// Mitsubishi GX Works2 project: PLC_group4 (1)   PLC: FX3G

// global labels: Global1
VAR_GLOBAL
  Start_Day_Switch AT X007 : BOOL;
  Oat_input AT D1110 : REAL;
  Oat_On_Hand AT D1120 : REAL;
  Protein_input AT D1130 : REAL;
  Protein_On_Hand AT D1140 : REAL;
  Honey_input AT D1150 : REAL;
  Honey_On_Hand AT D1160 : REAL;
END_VAR
VAR_GLOBAL CONSTANT
  Oat_LB : REAL := 400.0;
  Honey_LB : REAL := 160.0;
END_VAR
VAR_GLOBAL
  Ready_for_production AT M0 : BOOL;
  Emergency_Switch AT X005 : BOOL;
  Day_On AT Y000 : BOOL;
  Choose_Type AT X003 : BOOL;
  Analog_input1 AT D8280 : INT;
END_VAR
VAR_GLOBAL CONSTANT
  divide_input : REAL := 400.0;
  Protein_LB1 : REAL := 320.0;
END_VAR
VAR_GLOBAL
  Analog1_value AT D1170 : REAL;
END_VAR
VAR_GLOBAL CONSTANT
  Protein_type_LB : REAL := 5;
END_VAR
VAR_GLOBAL
  Protein_indicator AT M4 : BOOL;
END_VAR
VAR_GLOBAL CONSTANT
  Calssic_type_UB : REAL := 5.0;
END_VAR
VAR_GLOBAL
  Classic_indicator AT M5 : BOOL;
END_VAR
VAR_GLOBAL CONSTANT
  Oat_Classic_LB : REAL := 400.0;
  Protein_pro_LB1 : REAL := 320.0;
  Honey_pro_LB : REAL := 160.0;
END_VAR
VAR_GLOBAL
  Flag_oatClassic_production AT M1 : BOOL;
  Flag_proteinPro_production AT M2 : BOOL;
  Flag_honeyPro_production AT M3 : BOOL;
END_VAR
VAR_GLOBAL CONSTANT
  Protein_Calssic_LB : REAL := 160.0;
END_VAR
VAR_GLOBAL
  Flag_proteinClassic_production AT M6 : BOOL;
END_VAR
VAR_GLOBAL CONSTANT
  Honey_Classic_LB : REAL := 120.0;
END_VAR
VAR_GLOBAL
  Flag_HoneyClassic_production AT M7 : BOOL;
  Classic_check AT M8 : BOOL;
END_VAR
VAR_GLOBAL CONSTANT
  Oat_protein_LB : REAL := 240.0;
END_VAR
VAR_GLOBAL
  Flag_oatPro_production AT M9 : BOOL;
  Pro_check AT M10 : BOOL;
  TimerPro AT TC1 : BOOL;
  TV_5sec AT K50 : WORD;
  Mixing AT Y003 : BOOL;
  Stat_mix AT TS1 : BOOL;
  Analog_Output1 AT D8282 : INT;
  energy_bar_amount AT D1100 : REAL;
END_VAR
VAR_GLOBAL CONSTANT
  Mix_Classic : REAL := 680;
END_VAR
VAR_GLOBAL
  Mix_Total AT D1190 : REAL;
END_VAR
VAR_GLOBAL CONSTANT
  Mix_Pro : REAL := 720;
END_VAR
VAR_GLOBAL
  Start_Cooking AT X002 : BOOL;
  finish_cooking AT M11 : BOOL;
  help_cook AT M12 : BOOL;
  TC_2 AT TC2 : BOOL;
  blinkTime AT K5 : WORD;
  TS_2 AT TS2 : BOOL;
  Y_1 AT Y001 : BOOL;
  TC_3 AT TC3 : BOOL;
  TS_3 AT TS3 : BOOL;
  Y_2 AT Y002 : BOOL;
  TC_4 AT TC4 : BOOL;
  Classic_Time AT K40 : WORD;
  Protein_Time AT K50 : WORD;
  TC_5 AT TC5 : BOOL;
  Cooking_Tot AT D1200 : REAL;
  TS_4 AT TS4 : BOOL;
  TS_5 AT TS5 : BOOL;
  Start_pack AT X006 : BOOL;
  This_pack AT X000 : BOOL;
  One_packed AT K1 : WORD;
  One_start AT CC1 : BOOL;
  Eight_end AT CC2 : BOOL;
  Eight_packed AT K8 : WORD;
  Add_pack AT CS1 : BOOL;
  Last_pack AT CS2 : BOOL;
  Pack_inProcess AT Y004 : BOOL;
  Total_packges AT D1210 : REAL;
  Add_packge AT E1.0 : REAL;
END_VAR
VAR_GLOBAL CONSTANT
  Change_to_double : REAL := 40.0;
END_VAR
VAR_GLOBAL
  TS_1 AT TS1 : BOOL;
  finish_mix AT M13 : BOOL;
END_VAR

// task Task_01 (event TRUE, interval 0, priority 31): POU_01

PROGRAM POU_01
VAR CONSTANT
  Protein_LB : REAL := 320.0;
END_VAR
VAR
  analog_output : WORD;
END_VAR
(* structured ladder/FBD written out as ST: instructions are called as NAME(EN, inputs, outputs); _pN, _eN, _tN stand for wires *)
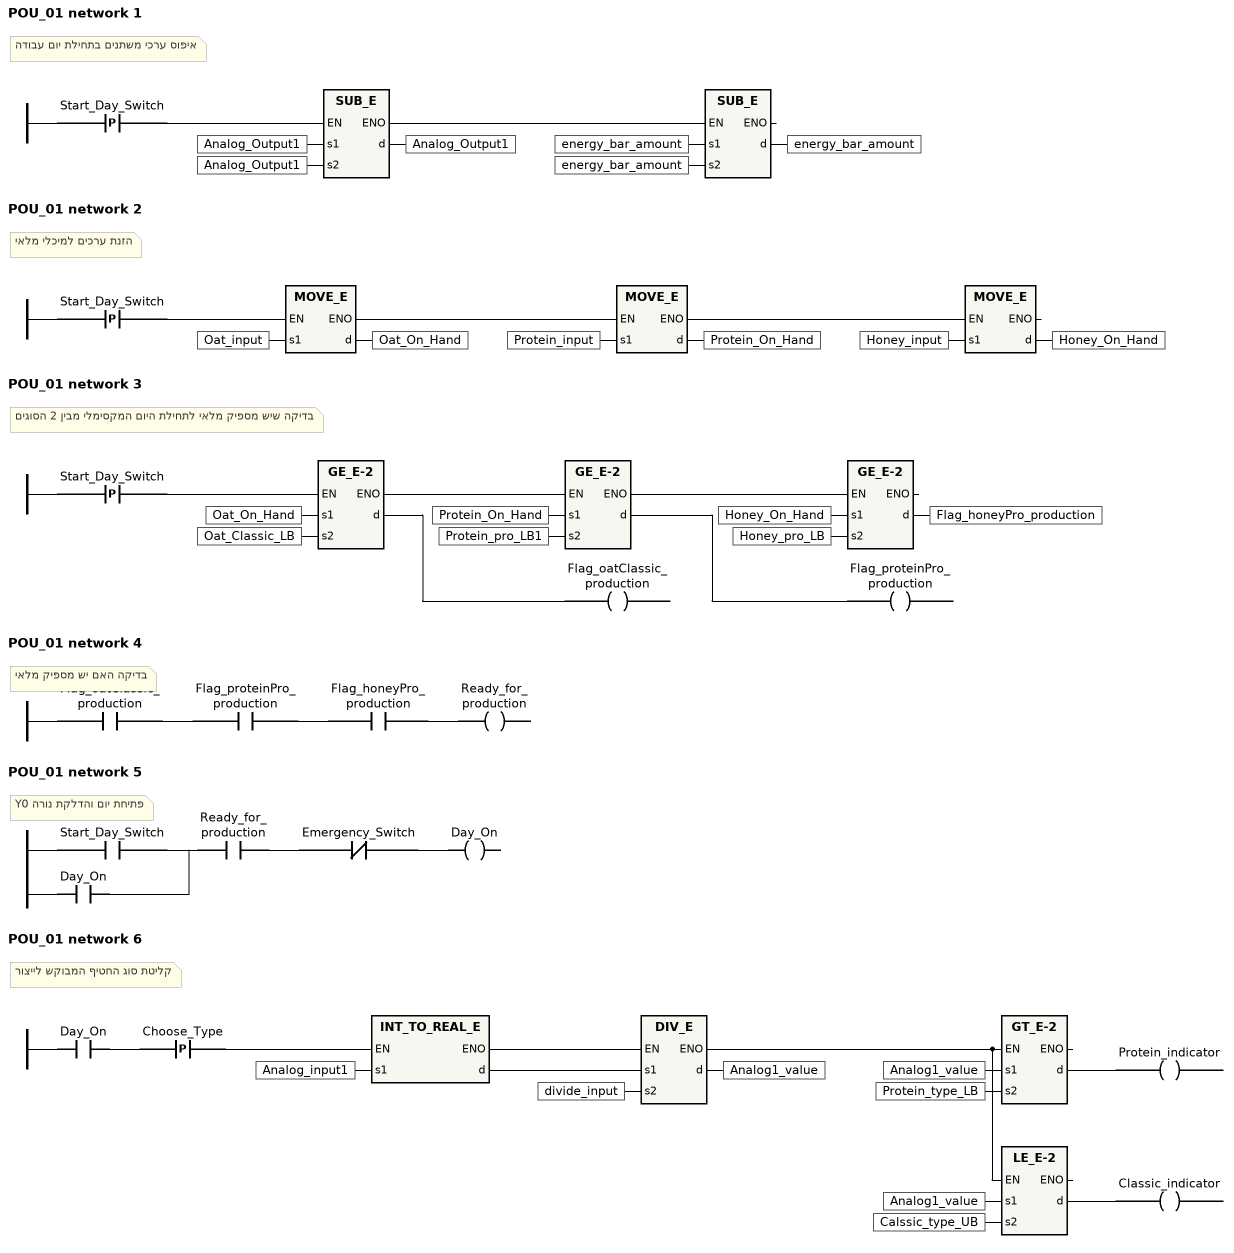
(* network 1 *)
(* איפוס ערכי משתנים בתחילת יום עבודה *)
_e1 := SUB_E(LDP(TRUE, Start_Day_Switch), Analog_Output1, Analog_Output1, Analog_Output1);
SUB_E(_e1, energy_bar_amount, energy_bar_amount, energy_bar_amount);
(* network 2 *)
(* הזנת ערכים למיכלי מלאי *)
_e1 := MOVE_E(LDP(TRUE, Start_Day_Switch), Oat_input, Oat_On_Hand);
_e2 := MOVE_E(_e1, Protein_input, Protein_On_Hand);
MOVE_E(_e2, Honey_input, Honey_On_Hand);
(* network 3 *)
(* בדיקה שיש מספיק מלאי לתחילת היום המקסימלי מבין 2 הסוגים *)
_e2 := GE_E(LDP(TRUE, Start_Day_Switch), Oat_On_Hand, Oat_Classic_LB, _t1);
_e4 := GE_E(_e2, Protein_On_Hand, Protein_pro_LB1, _t3);
GE_E(_e4, Honey_On_Hand, Honey_pro_LB, Flag_honeyPro_production);
Flag_oatClassic_production := _t1;
Flag_proteinPro_production := _t3;
(* network 4 *)
(* בדיקה האם יש מספיק מלאי *)
Ready_for_production := Flag_oatClassic_production AND Flag_proteinPro_production AND Flag_honeyPro_production;
(* network 5 *)
(* פתיחת יום והדלקת נורה Y0 *)
Day_On := ((Start_Day_Switch OR Day_On) AND Ready_for_production) AND NOT Emergency_Switch;
(* network 6 *)
(* קליטת סוג החטיף המבוקש לייצור *)
_e2 := INT_TO_REAL_E(Day_On AND LDP(TRUE, Choose_Type), Analog_input1, _t1);
_e3 := DIV_E(_e2, _t1, divide_input, Analog1_value);
GT_E(_e3, Analog1_value, Protein_type_LB, _t4);
Protein_indicator := _t4;
LE_E(_e3, Analog1_value, Calssic_type_UB, _t5);
Classic_indicator := _t5;
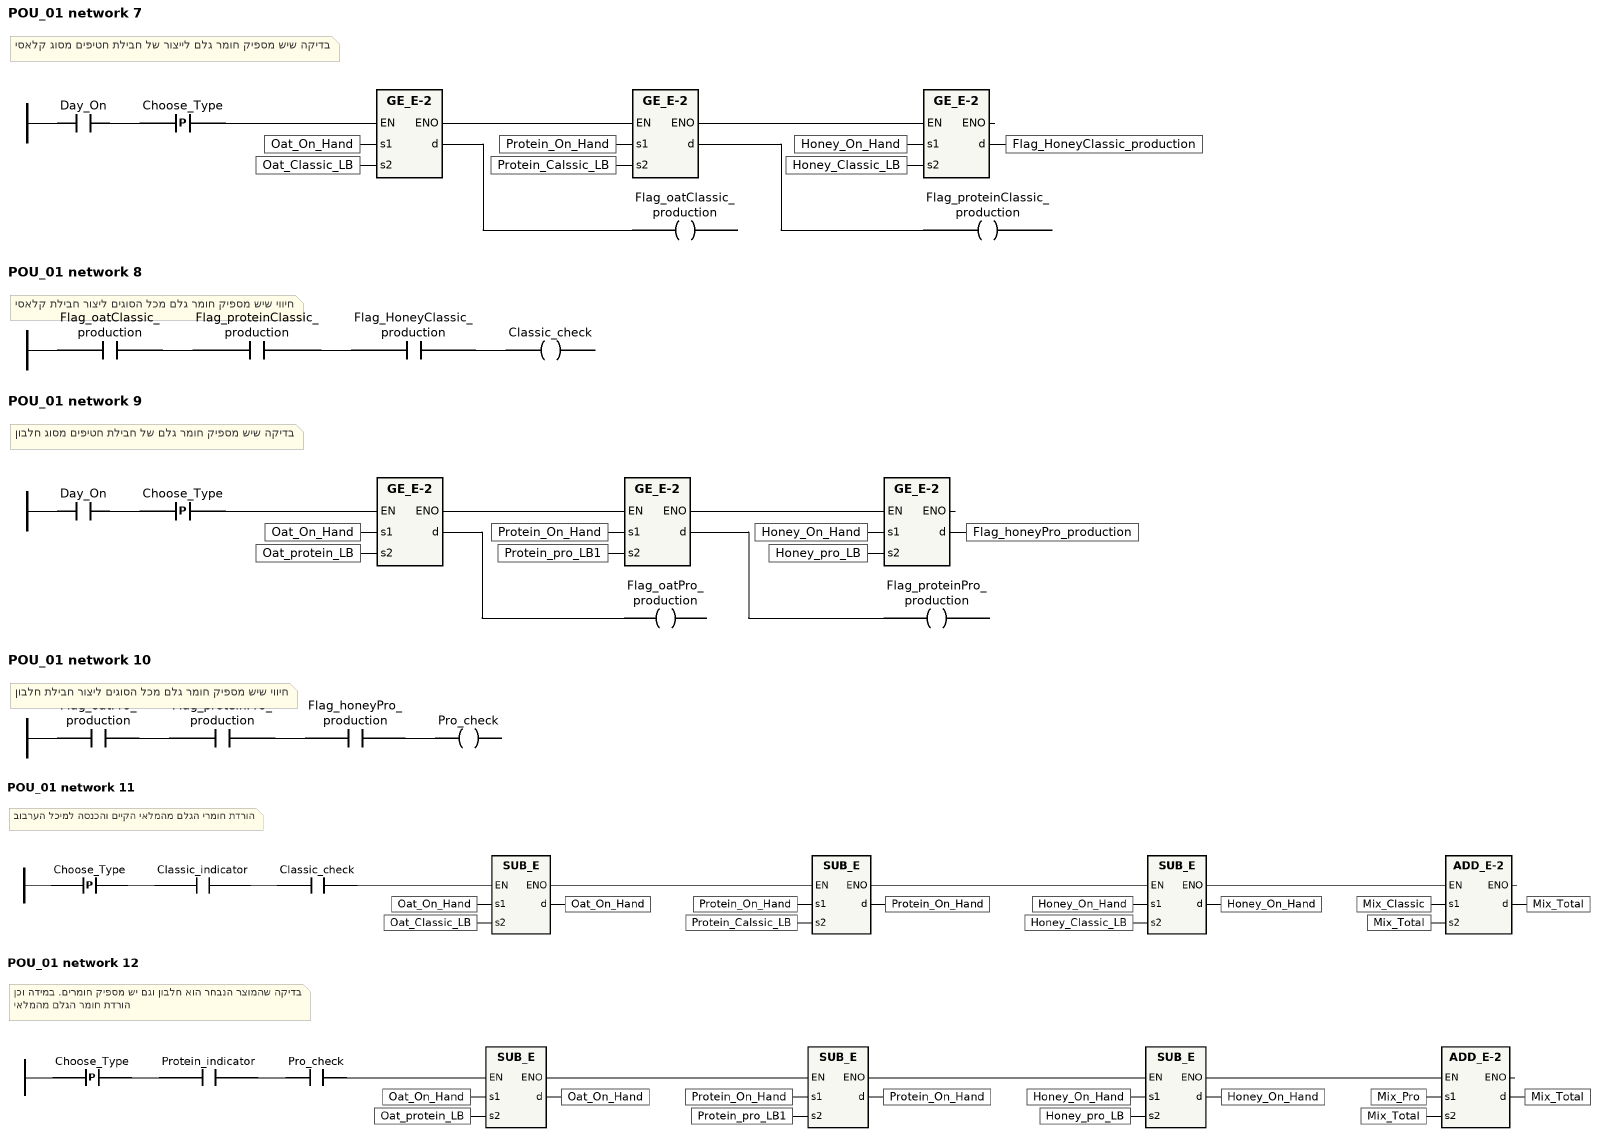
(* network 7 *)
(* בדיקה שיש מספיק חומר גלם לייצור של חבילת חטיפים מסוג קלאסי *)
_e2 := GE_E(Day_On AND LDP(TRUE, Choose_Type), Oat_On_Hand, Oat_Classic_LB, _t1);
_e4 := GE_E(_e2, Protein_On_Hand, Protein_Calssic_LB, _t3);
GE_E(_e4, Honey_On_Hand, Honey_Classic_LB, Flag_HoneyClassic_production);
Flag_proteinClassic_production := _t3;
Flag_oatClassic_production := _t1;
(* network 8 *)
(* חיווי שיש מספיק חומר גלם מכל הסוגים ליצור חבילת קלאסי *)
Classic_check := Flag_oatClassic_production AND Flag_proteinClassic_production AND Flag_HoneyClassic_production;
(* network 9 *)
(* בדיקה שיש מספיק חומר גלם של חבילת חטיפים מסוג חלבון *)
_e2 := GE_E(Day_On AND LDP(TRUE, Choose_Type), Oat_On_Hand, Oat_protein_LB, _t1);
_e4 := GE_E(_e2, Protein_On_Hand, Protein_pro_LB1, _t3);
GE_E(_e4, Honey_On_Hand, Honey_pro_LB, Flag_honeyPro_production);
Flag_proteinPro_production := _t3;
Flag_oatPro_production := _t1;
(* network 10 *)
(* חיווי שיש מספיק חומר גלם מכל הסוגים ליצור חבילת חלבון *)
Pro_check := Flag_oatPro_production AND Flag_proteinPro_production AND Flag_honeyPro_production;
(* network 11 *)
(* הורדת חומרי הגלם מהמלאי הקיים והכנסה למיכל הערבוב *)
_e1 := SUB_E(LDP(TRUE, Choose_Type) AND Classic_indicator AND Classic_check, Oat_On_Hand, Oat_Classic_LB, Oat_On_Hand);
_e2 := SUB_E(_e1, Protein_On_Hand, Protein_Calssic_LB, Protein_On_Hand);
_e3 := SUB_E(_e2, Honey_On_Hand, Honey_Classic_LB, Honey_On_Hand);
ADD_E(_e3, Mix_Classic, Mix_Total, Mix_Total);
(* network 12 *)
(* בדיקה שהמוצר הנבחר הוא חלבון וגם יש מספיק חומרים. במידה וכן הורדת חומר הגלם מהמלאי *)
_e1 := SUB_E(LDP(TRUE, Choose_Type) AND Protein_indicator AND Pro_check, Oat_On_Hand, Oat_protein_LB, Oat_On_Hand);
_e2 := SUB_E(_e1, Protein_On_Hand, Protein_pro_LB1, Protein_On_Hand);
_e3 := SUB_E(_e2, Honey_On_Hand, Honey_pro_LB, Honey_On_Hand);
ADD_E(_e3, Mix_Pro, Mix_Total, Mix_Total);
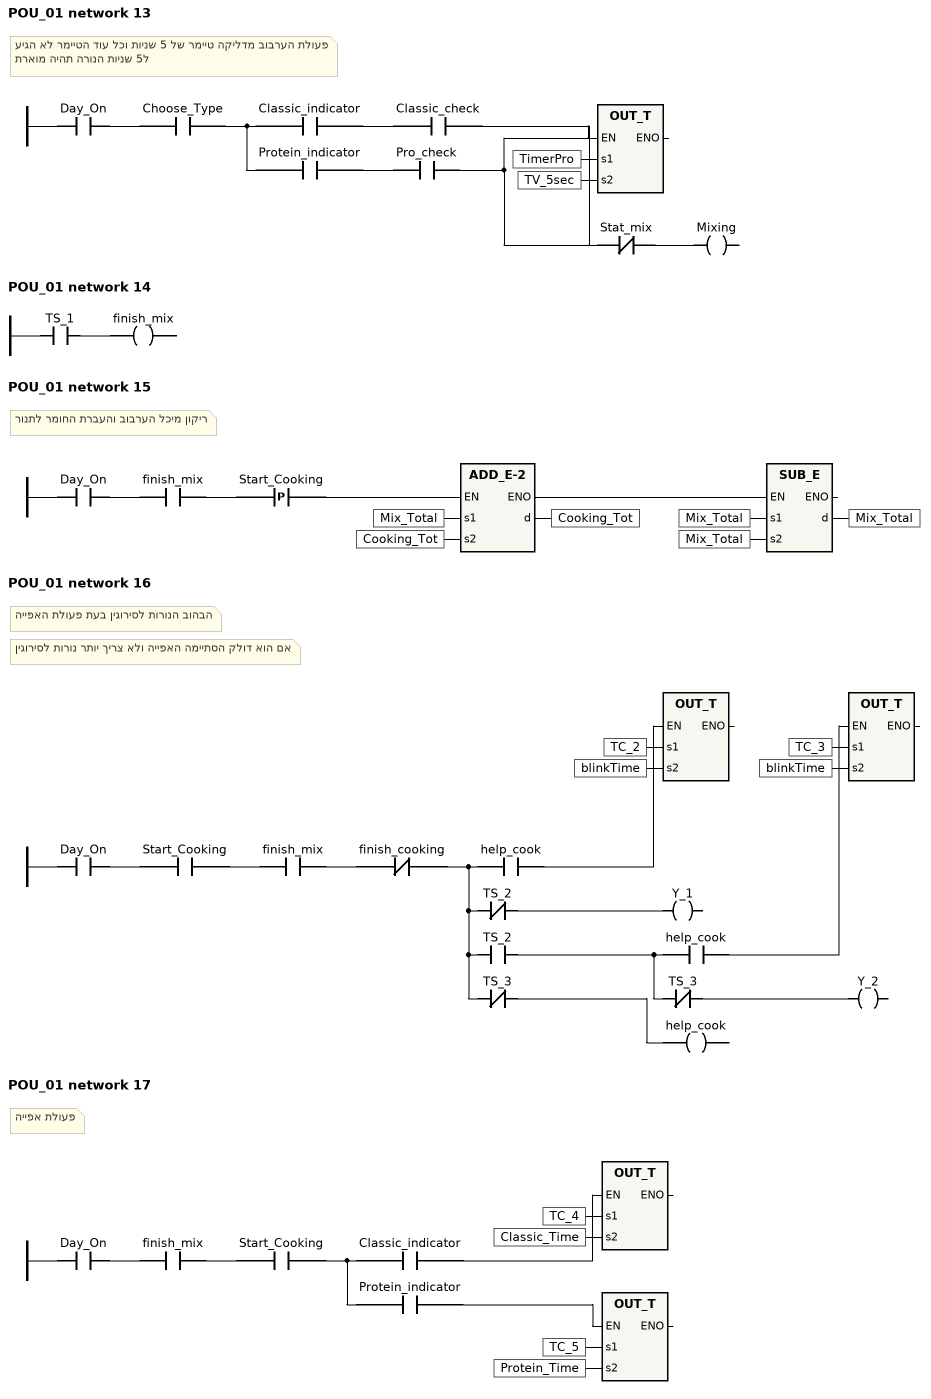
(* network 13 *)
(* פעולת הערבוב מדליקה טיימר של 5 שניות וכל עוד הטיימר לא הגיע ל5 שניות הנורה תהיה מוארת *)
_p1 := Day_On AND Choose_Type;
_p2 := (_p1 AND Classic_indicator AND Classic_check) OR (_p1 AND Protein_indicator AND Pro_check);
Mixing := _p2 AND NOT Stat_mix;
OUT_T(_p2, TimerPro, TV_5sec);
(* network 14 *)
finish_mix := TS_1;
(* network 15 *)
(* ריקון מיכל הערבוב והעברת החומר לתנור *)
_e1 := ADD_E(Day_On AND finish_mix AND LDP(TRUE, Start_Cooking), Mix_Total, Cooking_Tot, Cooking_Tot);
SUB_E(_e1, Mix_Total, Mix_Total, Mix_Total);
(* network 16 *)
(* הבהוב הנורות לסירוגין בעת פעולת האפייה *)
(* אם הוא דולק הסתיימה האפייה ולא צריך יותר נורות לסירוגין *)
_p1 := Day_On AND Start_Cooking AND finish_mix AND NOT finish_cooking;
OUT_T(_p1 AND help_cook, TC_2, blinkTime);
Y_1 := _p1 AND NOT TS_2;
_p2 := _p1 AND TS_2;
OUT_T(_p2 AND help_cook, TC_3, blinkTime);
Y_2 := _p2 AND NOT TS_3;
help_cook := _p1 AND NOT TS_3;
(* network 17 *)
(* פעולת אפייה *)
_p1 := Day_On AND finish_mix AND Start_Cooking;
OUT_T(_p1 AND Classic_indicator, TC_4, Classic_Time);
OUT_T(_p1 AND Protein_indicator, TC_5, Protein_Time);
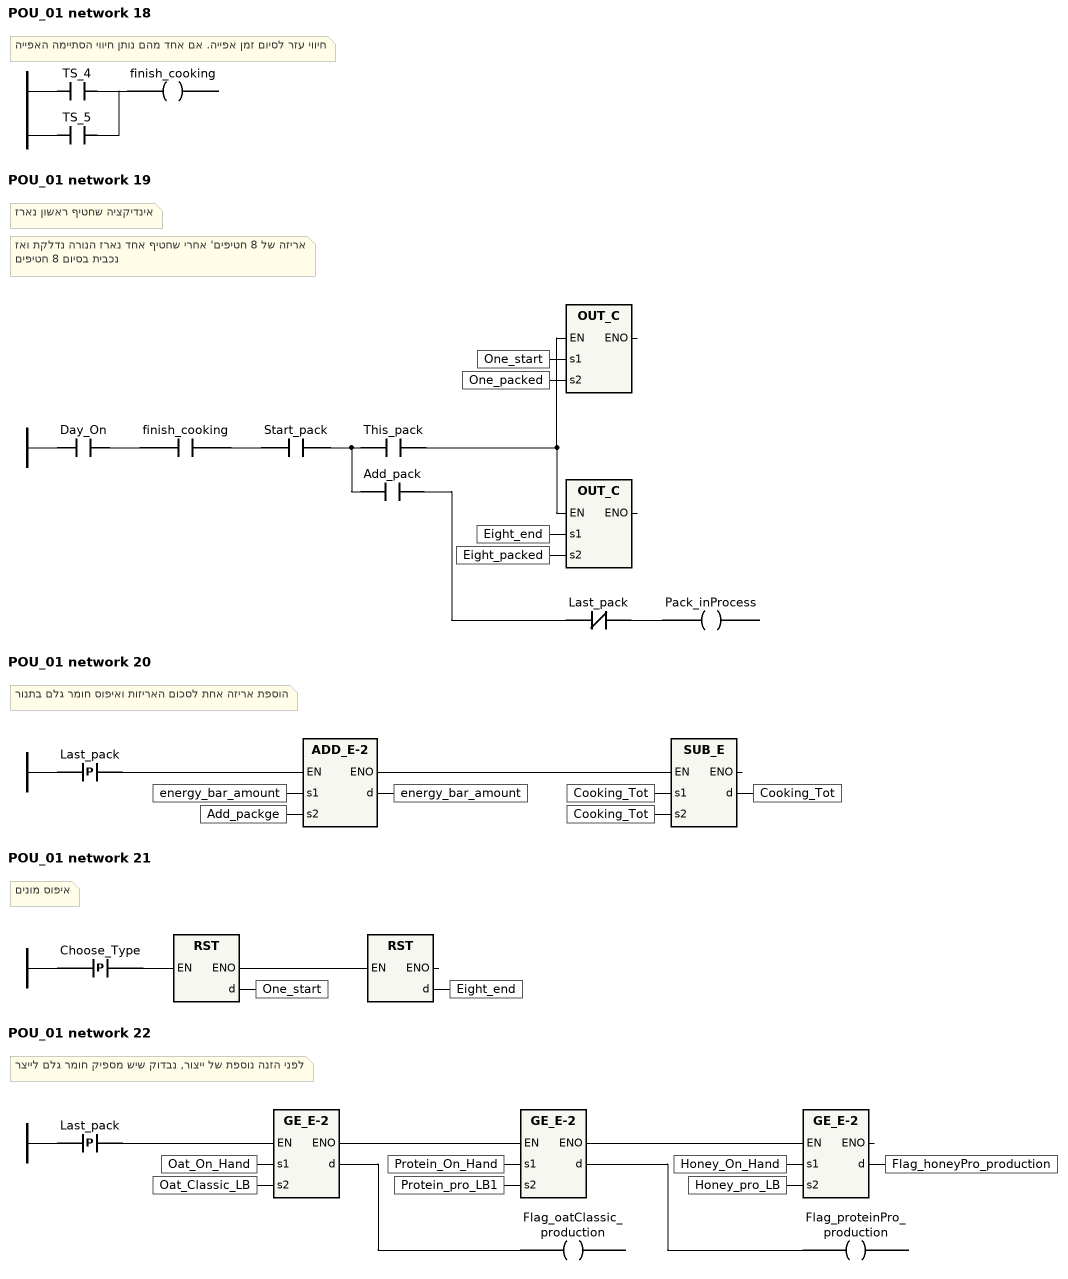
(* network 18 *)
(* חיווי עזר לסיום זמן אפייה. אם אחד מהם נותן חיווי הסתיימה האפייה *)
finish_cooking := TS_4 OR TS_5;
(* network 19 *)
(* אינדיקציה שחטיף ראשון נארז *)
(* אריזה של 8 חטיפים' אחרי שחטיף אחד נארז הנורה נדלקת ואז נכבית בסיום 8 חטיפים *)
_p1 := Day_On AND finish_cooking AND Start_pack;
_p2 := _p1 AND This_pack;
OUT_C(_p2, One_start, One_packed);
OUT_C(_p2, Eight_end, Eight_packed);
Pack_inProcess := _p1 AND Add_pack AND NOT Last_pack;
(* network 20 *)
(* הוספת אריזה אחת לסכום האריזות ואיפוס חומר גלם בתנור *)
_e1 := ADD_E(LDP(TRUE, Last_pack), energy_bar_amount, Add_packge, energy_bar_amount);
SUB_E(_e1, Cooking_Tot, Cooking_Tot, Cooking_Tot);
(* network 21 *)
(* איפוס מונים *)
_e1 := RST(LDP(TRUE, Choose_Type), One_start);
RST(_e1, Eight_end);
(* network 22 *)
(* לפני הזנה נוספת של ייצור, נבדוק שיש מספיק חומר גלם לייצר *)
_e2 := GE_E(LDP(TRUE, Last_pack), Oat_On_Hand, Oat_Classic_LB, _t1);
_e4 := GE_E(_e2, Protein_On_Hand, Protein_pro_LB1, _t3);
GE_E(_e4, Honey_On_Hand, Honey_pro_LB, Flag_honeyPro_production);
Flag_oatClassic_production := _t1;
Flag_proteinPro_production := _t3;
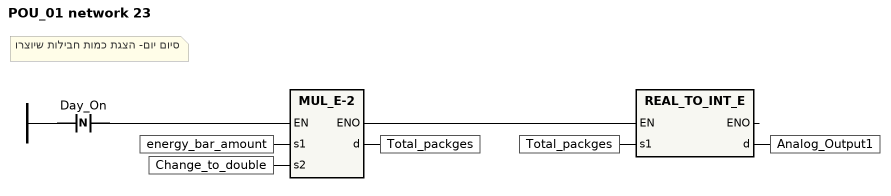
(* network 23 *)
(* סיום יום- הצגת כמות חבילות שיוצרו *)
_e1 := MUL_E(LDF(TRUE, Day_On), energy_bar_amount, Change_to_double, Total_packges);
REAL_TO_INT_E(_e1, Total_packges, Analog_Output1);
END_PROGRAM
